ABB RobotStudio station: Lab1Part1.rspag

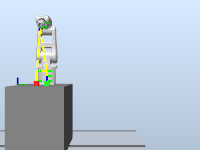
--- station ---
Station PickAndPlace (saved by RobotStudio 7.0.8732.594)
Controller IRB_120_PickAndPlace, task T_ROB1: task frame (RAPID world) sits at (-250, 0, 600) mm in the station
Controller IRB_120_PickAndPlace
  mechanical unit ROB_1: IRB120_3_58__01, 6 joints, base frame (0, 0, 0) mm
Layout (positions relative to the parent item):
  - RobotTable [part]
  - Workstation [part]
  - IRB120_3_58__01 [mechanism, from Robots\IRB120_3_58_G_01.rslib] at (-250, 0, 600) mm; joint values [0, 0, 0, 0, 0.5236, 0] (rad or m)
  - Smart_Gripper_Servo_Fingers [mechanism, from Libraries\Smart_Gripper_Servo_Fingers.rslib] at (114.35, 0, 1194) mm, rotated rx 180 ry 60 rz 180 deg; joint values [0.025] (rad or m)
  - TopPart [part]
  - BottomPart [part]
Attachment: Smart_Gripper_Servo_Fingers is attached to IRB120_3_58__01 / Link6
EventTableEntry 1039: Group=, Trigger=Gripper 1040, Actions=[EventTableActionMechanicalPose 1041, EventTableActionAttach 1114], Comment=, ActivationMode=2, Cyclic=false
EventTableTriggerIO 1040: IOValue=[1], IRC5Controller=? -1, Operator=0, SignalSource=IRB_120_PickAndPlace 515
EventTableActionMechanicalPose 1041: VirtualSignal=, Mechanism=Smart_Gripper_Servo_Fingers 1010, ToPoseName=SyncPosition, VirtualSignalValue=[1]
EventTableActionAttach 1114: AttachmentParent=Smart_Gripper_Servo_Fingers 1010, AttachmentChild=? -1, MountObject=false, Offset=[X=1, Y=0, Z=0, W=0, X=0, Y=1, Z=0, W=0, X=0, Y=0, Z=1, W=0, X=0, Y=0, Z=0, W=1], FlangeIndext=0, FindNearest=true
EventTableEntry 1115: Group=, Trigger=Gripper 1116, Actions=[EventTableActionMechanicalPose 1117, EventTableActionDetach 1118], Comment=, ActivationMode=2, Cyclic=false
EventTableTriggerIO 1116: IOValue=[0], IRC5Controller=? -1, Operator=0, SignalSource=IRB_120_PickAndPlace 515
EventTableActionMechanicalPose 1117: VirtualSignal=, Mechanism=Smart_Gripper_Servo_Fingers 1010, ToPoseName=HomePosition, VirtualSignalValue=[1]
EventTableActionDetach 1118: AttachmentParent=Smart_Gripper_Servo_Fingers 1010, AttachmentChild=? -1
Targets, tools, work objects and paths stored in the station and not in the controller backup, written as RAPID:
! task T_ROB1
MODULE Module1
  CONST robtarget Target_40:=[[250,320,45],[0,0,1,0],[0,0,0,0],[9E+09,9E+09,9E+09,9E+09,9E+09,9E+09]];
ENDMODULE


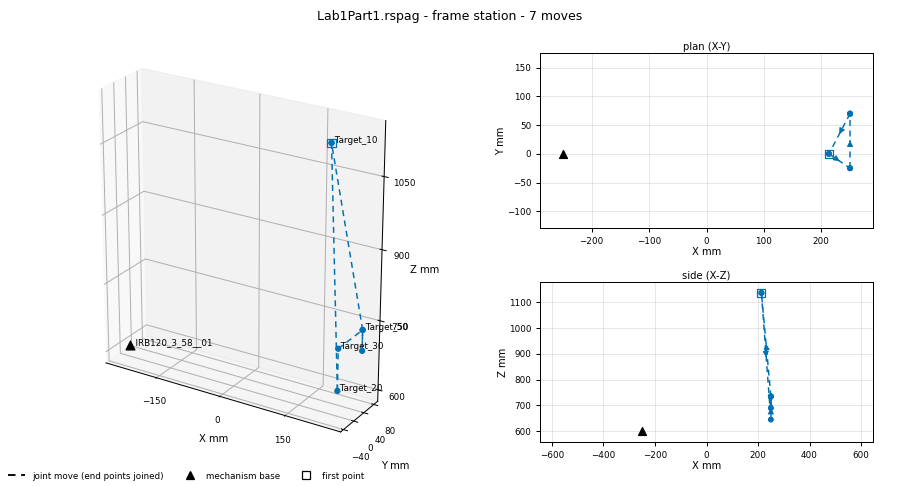
[picture p0: tool path of Lab1Part1.rspag in frame station, 7 of 7 moves have a stored position in this frame; points joined in program order, loops and branches not executed]
--- Backups/IRB_120_PickAndPlace/RAPID/TASK1/PROGMOD/CalibData.mod ---
MODULE CalibData
	PERS tooldata Servo:=[TRUE,[[0,0,114.2],[1,0,0,0]],[0.215,[8.7,12.3,49.2],[1,0,0,0],0.00021,0.00024,0.00009]];
	TASK PERS wobjdata Workobject_1:=[FALSE,TRUE,"",[[250,-250,0],[1,0,0,0]],[[0,0,0],[1,0,0,0]]];
ENDMODULE

--- Backups/IRB_120_PickAndPlace/RAPID/TASK1/PROGMOD/Module1.mod ---
MODULE Module1
	CONST robtarget Target_10:=[[463.253923279,0,536.899988039],[0.499999968,0,0.866025422,0],[0,0,0,0],[9E+09,9E+09,9E+09,9E+09,9E+09,9E+09]];
	CONST robtarget Target_20:=[[250,225,45],[0,0,1,0],[0,0,0,0],[9E+09,9E+09,9E+09,9E+09,9E+09,9E+09]];
	CONST robtarget Target_30:=[[250,225,135],[0,0,1,0],[0,0,0,0],[9E+09,9E+09,9E+09,9E+09,9E+09,9E+09]];
	CONST robtarget Target_50:=[[250,320,135],[0,0,1,0],[0,0,0,0],[9E+09,9E+09,9E+09,9E+09,9E+09,9E+09]];
	CONST robtarget Target_50_2:=[[250,320,90],[0,0,1,0],[0,0,0,0],[9E+09,9E+09,9E+09,9E+09,9E+09,9E+09]];
    !***********************************************************
    !
    ! Module:  Module1
    !
    ! Description:
    !   <Insert description here>
    !
    ! Author: bruno
    !
    ! Version: 1.0
    !
    !***********************************************************


    !***********************************************************
    !
    ! Procedure main
    !
    !   This is the entry point of your program
    !
    !***********************************************************
    PROC main()
        !Add your code here
    ENDPROC
	PROC Path_10()
	    Reset Gripper;
	    MoveJ Target_10,v100,z5,Servo\WObj:=wobj0;
	    MoveJ Target_20,v100,z5,Servo\WObj:=Workobject_1;
	    WaitTime\InPos,1;
	    Set Gripper;
	    MoveJ Target_30,v100,z5,Servo\WObj:=Workobject_1;
	    MoveJ Target_50,v100,z5,Servo\WObj:=Workobject_1;
	    MoveJ Target_50_2,v100,z5,Servo\WObj:=Workobject_1;
	    WaitTime\InPos,1;
	    Reset Gripper;
	    MoveJ Target_50,v100,z5,Servo\WObj:=Workobject_1;
	    MoveJ Target_10,v100,z5,Servo\WObj:=wobj0;
	ENDPROC
ENDMODULE

--- Backups/IRB_120_PickAndPlace/SYSPAR/EIO.cfg ---
EIO:CFG_1.0:6:1::
#
EIO_SIGNAL:

      -Name "Gripper" -SignalType "DO" -Access "All"
